# B&R Automation Studio project Pract2
Automation Studio 4.5.2.102; technology packages: mappMotion 5.2.1

## Configuration Config1

### Task classes (Cpu.sw)
```
Cyclic#4:
  Program <- Program.prg
VcDataObjects: Visu <- Visu.dob
Libraries: McBase
```

### Hardware
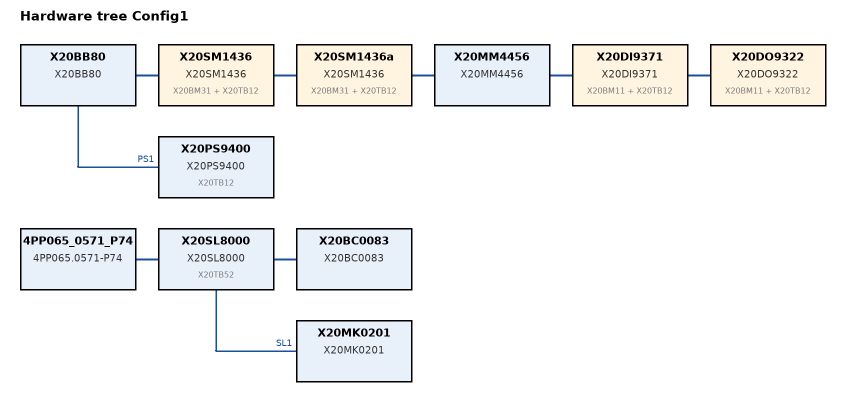
```
4PP065_0571_P74 : 4PP065.0571-P74 v1.1.2.0
  Connector IF5:
    ActivateDevice = 1
    Mode = Manual
    InternetAddress = 10.0.1.11
    SubnetMask = 255.255.255.0
  ConfigurationID = labBR
  VcObjectName = Visu
X20BB80 : X20BB80 v1.0.2.0
X20BC0083 : X20BC0083 v2.9.0.0  [PLK1 -> X20SL8000.PLK2 [Cable Type=PowerlinkCable, Length=10, Version=1.0.0.2]; SL -> X20BB80.SL1]
X20BM11 : X20BM11 v1.0.0.1  [X2X1 -> X20MM4456.X2X2]
X20BM11a : X20BM11 v1.0.0.1  [X2X1 -> X20BM11.X2X2]
X20BM31 : X20BM31 v1.0.0.1  [X2X1 -> X20BB80.IF1]
X20BM31a : X20BM31 v1.0.0.1  [X2X1 -> X20BM31.X2X2]
X20DI9371 : X20DI9371 v1.0.2.0  [SS1 -> X20TB12d.SS; SL -> X20BM11.SL1]
X20DO9322 : X20DO9322 v1.0.3.0  [SS1 -> X20TB12e.SS; SL -> X20BM11a.SL1]
X20MK0201 : X20MK0201 v1.0.0.0  [SL -> X20SL8000.SL1]
X20MM4456 : X20MM4456 v1.1.5.0  [X2X1 -> X20BM31a.X2X2]
X20PS9400 : X20PS9400 v1.0.2.4  [SS1 -> X20TB12.SS; PS -> X20BB80.PS1]
X20SL8000 : X20SL8000 v1.6.5.2  [PLK1 -> 4PP065_0571_P74.IF4 [Cable Type=PowerlinkCable, Length=10, Version=1.0.0.2]; PLK2 -> X20BC0083.PLK1 [Cable Type=PowerlinkCable, Length=10, Version=1.0.0.2]; SS1 -> X20TB52.SS]
  SafeProject = SafeLOGIC-1
X20SM1436 : X20SM1436 v2.2.0.0  [SS1 -> X20TB12b.SS; SL -> X20BM31.SL1]
X20SM1436a : X20SM1436 v2.2.0.0  [SS1 -> X20TB12c.SS; SL -> X20BM31a.SL1]
X20TB12 : X20TB12 v1.0.0.0
X20TB12b : X20TB12 v1.0.0.0
X20TB12c : X20TB12 v1.0.0.0
X20TB12d : X20TB12 v1.0.0.0
X20TB12e : X20TB12 v1.0.0.0
X20TB52 : X20TB52 v1.0.0.1
```

### IoMap.iom - 4PP065_0571_P74/IoMap.iom
```iecst
VAR_CONFIG
	::Program:LED[0] AT %QX."X20DO9322".DigitalOutput02;
	::Program:LED[1] AT %QX."X20DO9322".DigitalOutput03;
	::Program:LED[2] AT %QX."X20DO9322".DigitalOutput04;
	::Program:LED[3] AT %QX."X20DO9322".DigitalOutput05;
END_VAR
```

## Logical view

### Program Logical/Program (ANSIC)

#### Variables.var
```iecst
VAR
	LED : {REDUND_UNREPLICABLE} ARRAY[0..3] OF BOOL := [4(FALSE)];
	virtual_lamp : {REDUND_UNREPLICABLE} ARRAY[0..3] OF BOOL;
END_VAR
```

#### Main.c
```c
#include <bur/plctypes.h>

#ifdef _DEFAULT_INCLUDES
	#include <AsDefault.h>
#endif

void _INIT ProgramInit(void)
{

}

void _CYCLIC ProgramCyclic(void)
{
virtual_lamp[0]=LED[0];
virtual_lamp[1]=LED[1];
virtual_lamp[2]=LED[2];
virtual_lamp[3]=LED[3];

}

void _EXIT ProgramExit(void)
{

}
```

- Visualisation Logical/Visu (not shown)

Listed in the project but not available here: Logical/Global.typ, Logical/Global.var, Logical/Libraries
